PROGRAM Indicators
VAR
	TON_0: TON;
	TON_0_True: BOOL;
	TON_1: TON;
	TON_1_True: BOOL;
END_VAR

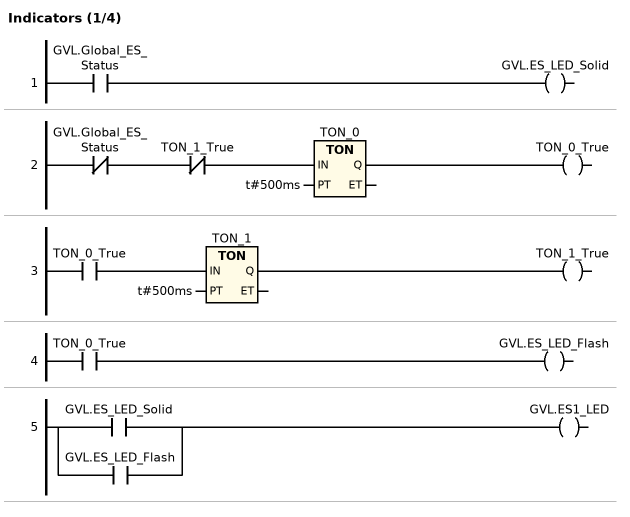
// NETWORK 1
GVL.ES_LED_Solid := GVL.Global_ES_Status;

// NETWORK 2
TON_0(IN := NOT GVL.Global_ES_Status AND NOT TON_1_True, PT := t#500ms); // TON
TON_0_True := TON_0.Q;

// NETWORK 3
TON_1(IN := TON_0_True, PT := t#500ms); // TON
TON_1_True := TON_1.Q;

// NETWORK 4
GVL.ES_LED_Flash := TON_0_True;

// NETWORK 5
GVL.ES1_LED := GVL.ES_LED_Solid OR GVL.ES_LED_Flash;

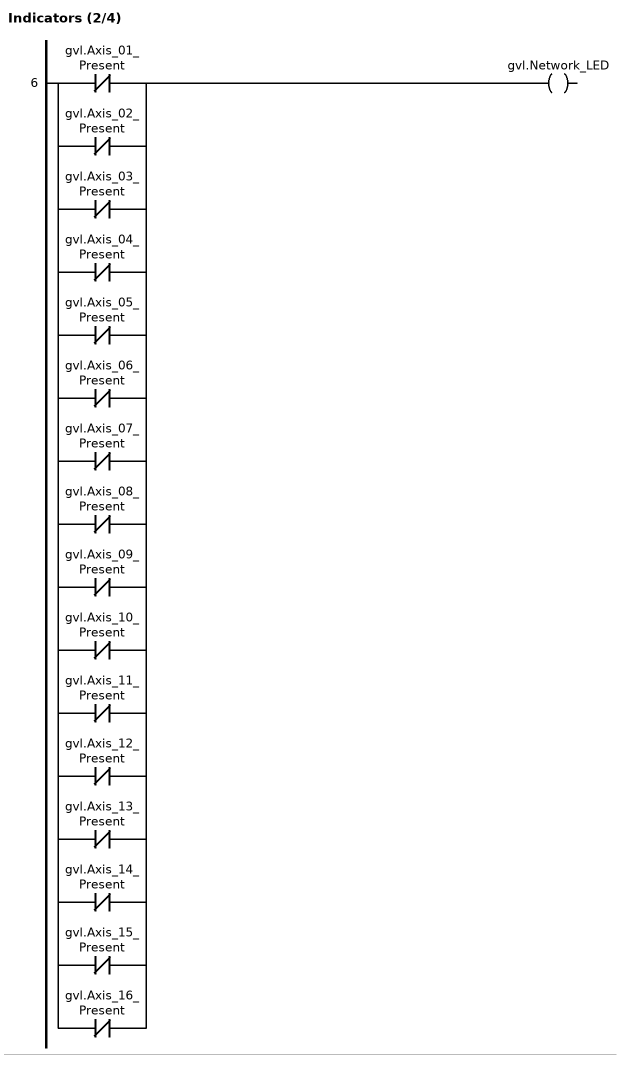
// NETWORK 6
gvl.Network_LED := NOT gvl.Axis_01_Present OR NOT gvl.Axis_02_Present OR NOT gvl.Axis_03_Present OR NOT gvl.Axis_04_Present OR NOT gvl.Axis_05_Present OR NOT gvl.Axis_06_Present OR NOT gvl.Axis_07_Present OR NOT gvl.Axis_08_Present OR NOT gvl.Axis_09_Present OR NOT gvl.Axis_10_Present OR NOT gvl.Axis_11_Present OR NOT gvl.Axis_12_Present OR NOT gvl.Axis_13_Present OR NOT gvl.Axis_14_Present OR NOT gvl.Axis_15_Present OR NOT gvl.Axis_16_Present;

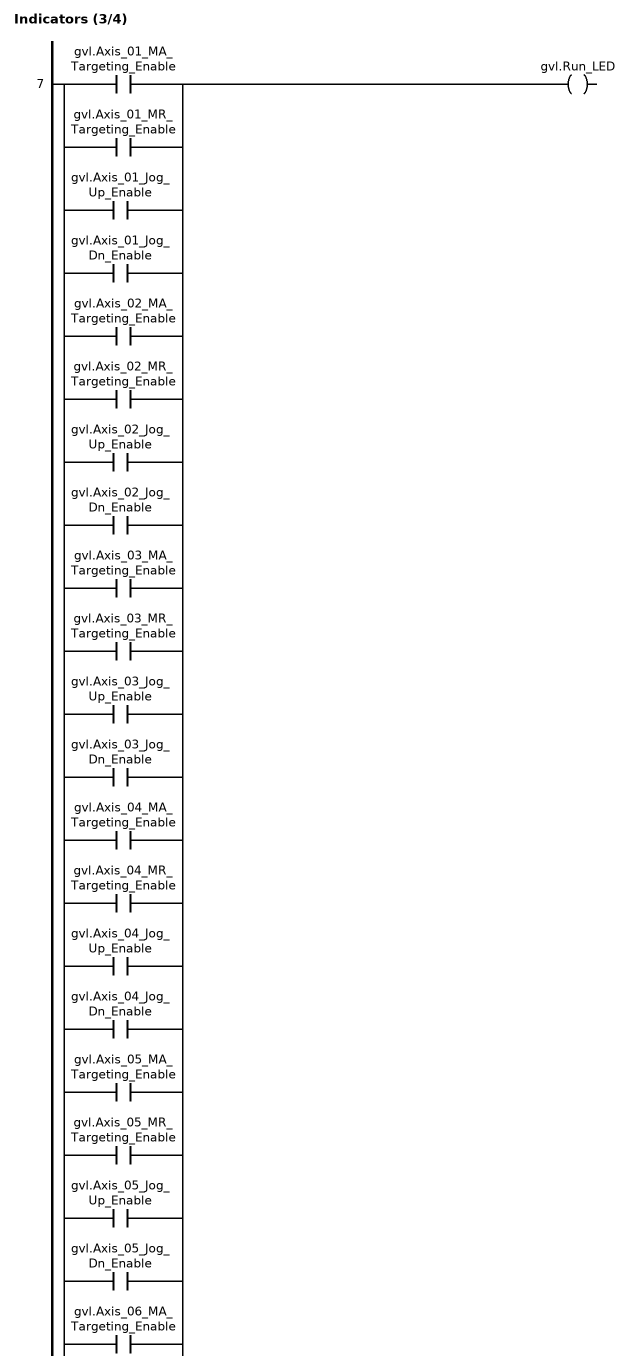
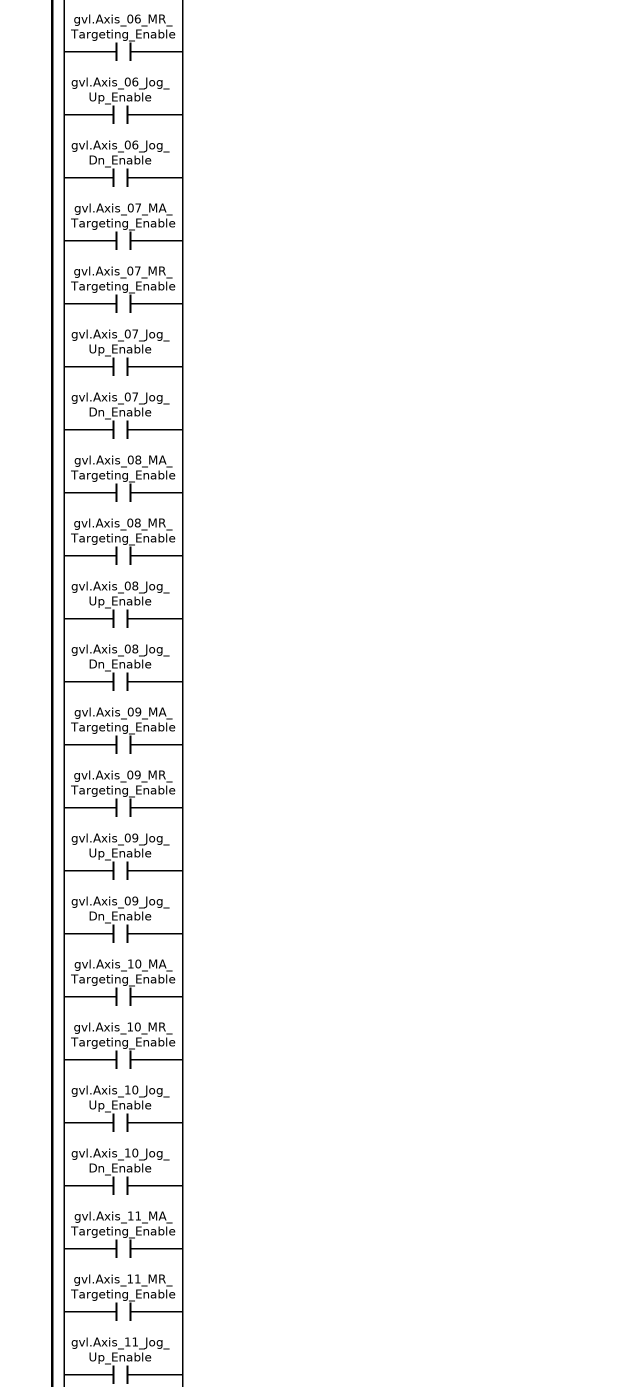
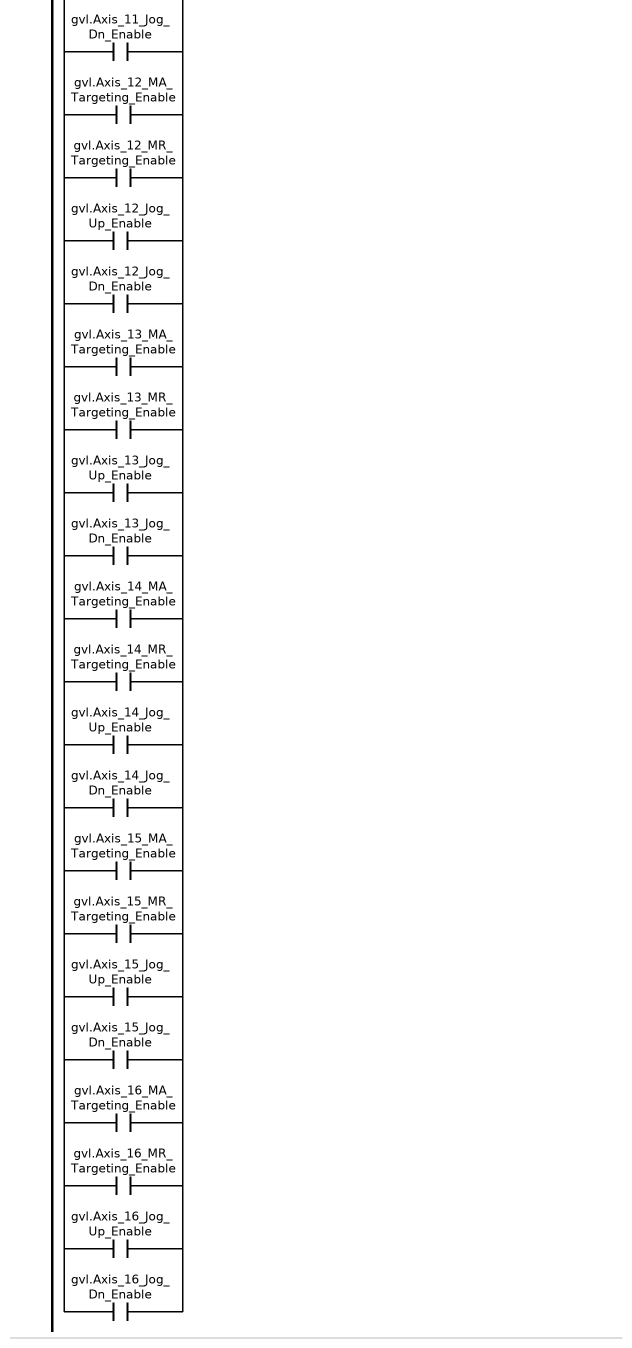
// NETWORK 7
gvl.Run_LED := gvl.Axis_01_MA_Targeting_Enable OR gvl.Axis_01_MR_Targeting_Enable OR gvl.Axis_01_Jog_Up_Enable OR gvl.Axis_01_Jog_Dn_Enable OR gvl.Axis_02_MA_Targeting_Enable OR gvl.Axis_02_MR_Targeting_Enable OR gvl.Axis_02_Jog_Up_Enable OR gvl.Axis_02_Jog_Dn_Enable OR gvl.Axis_03_MA_Targeting_Enable OR gvl.Axis_03_MR_Targeting_Enable OR gvl.Axis_03_Jog_Up_Enable OR gvl.Axis_03_Jog_Dn_Enable OR gvl.Axis_04_MA_Targeting_Enable OR gvl.Axis_04_MR_Targeting_Enable OR gvl.Axis_04_Jog_Up_Enable OR gvl.Axis_04_Jog_Dn_Enable OR gvl.Axis_05_MA_Targeting_Enable OR gvl.Axis_05_MR_Targeting_Enable OR gvl.Axis_05_Jog_Up_Enable OR gvl.Axis_05_Jog_Dn_Enable OR gvl.Axis_06_MA_Targeting_Enable OR gvl.Axis_06_MR_Targeting_Enable OR gvl.Axis_06_Jog_Up_Enable OR gvl.Axis_06_Jog_Dn_Enable OR gvl.Axis_07_MA_Targeting_Enable OR gvl.Axis_07_MR_Targeting_Enable OR gvl.Axis_07_Jog_Up_Enable OR gvl.Axis_07_Jog_Dn_Enable OR gvl.Axis_08_MA_Targeting_Enable OR gvl.Axis_08_MR_Targeting_Enable OR gvl.Axis_08_Jog_Up_Enable OR gvl.Axis_08_Jog_Dn_Enable OR gvl.Axis_09_MA_Targeting_Enable OR gvl.Axis_09_MR_Targeting_Enable OR gvl.Axis_09_Jog_Up_Enable OR gvl.Axis_09_Jog_Dn_Enable OR gvl.Axis_10_MA_Targeting_Enable OR gvl.Axis_10_MR_Targeting_Enable OR gvl.Axis_10_Jog_Up_Enable OR gvl.Axis_10_Jog_Dn_Enable OR gvl.Axis_11_MA_Targeting_Enable OR gvl.Axis_11_MR_Targeting_Enable OR gvl.Axis_11_Jog_Up_Enable OR gvl.Axis_11_Jog_Dn_Enable OR gvl.Axis_12_MA_Targeting_Enable OR gvl.Axis_12_MR_Targeting_Enable OR gvl.Axis_12_Jog_Up_Enable OR gvl.Axis_12_Jog_Dn_Enable OR gvl.Axis_13_MA_Targeting_Enable OR gvl.Axis_13_MR_Targeting_Enable OR gvl.Axis_13_Jog_Up_Enable OR gvl.Axis_13_Jog_Dn_Enable OR gvl.Axis_14_MA_Targeting_Enable OR gvl.Axis_14_MR_Targeting_Enable OR gvl.Axis_14_Jog_Up_Enable OR gvl.Axis_14_Jog_Dn_Enable OR gvl.Axis_15_MA_Targeting_Enable OR gvl.Axis_15_MR_Targeting_Enable OR gvl.Axis_15_Jog_Up_Enable OR gvl.Axis_15_Jog_Dn_Enable OR gvl.Axis_16_MA_Targeting_Enable OR gvl.Axis_16_MR_Targeting_Enable OR gvl.Axis_16_Jog_Up_Enable OR gvl.Axis_16_Jog_Dn_Enable;

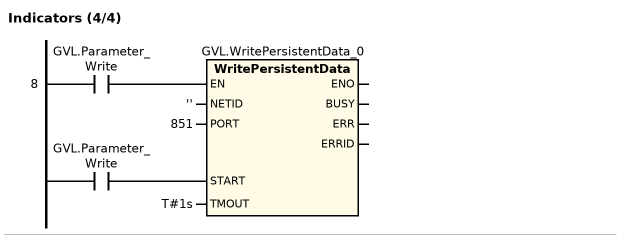
// NETWORK 8
IF GVL.Parameter_Write THEN
    GVL.WritePersistentData_0(NETID := '', PORT := 851, START := GVL.Parameter_Write, TMOUT := T#1s); // WritePersistentData
END_IF

END_PROGRAM

(* stored: Version 1.1.0.1, ProductVersion 3.1.4022.12
   POU Indicators: Id {2e086451-c4a9-40bd-b1d9-ee19be4226af}, SpecialFunc None *)
